(*
SPDX-FileCopyrightText: © 2026 Oleksandr Tiutyk <trofimich@gmail.com>
SPDX-License-Identifier: MIT
License: https://opensource.org/license/mit
*)

{attribute 'no_explicit_call' := 'do not call this function block directly'} 
FUNCTION_BLOCK GenericValueValidator EXTENDS Object IMPLEMENTS IGenericValueValidator
VAR
	_ClassName : STRING := __POUNAME();
	
	_TypeClass : GENERIC_TYPE_CLASS;
END_VAR

{attribute 'monitoring' := 'call'}
PROPERTY ClassName : REFERENCE TO STRING
GET
ClassName REF= _ClassName;
END_GET
END_PROPERTY

//!<param name="bInitRetains">if TRUE, the retain variables are initialized (warm start / cold start)</param>

//!<param name="bInCopyCode">if TRUE, the instance afterwards gets moved into the copy code (online change)</param>

METHOD FB_init : BOOL
VAR_INPUT
	
	bInitRetains	: BOOL;
	
	bInCopyCode	: BOOL;
	typeClass : GENERIC_TYPE_CLASS;
END_VAR
_TypeClass := typeClass;
END_METHOD

{attribute 'monitoring' := 'call'}
PROPERTY NamespaceName : REFERENCE TO STRING
GET
NamespaceName REF= CurrentNamespace.Name;
END_GET
END_PROPERTY

{attribute 'monitoring' := 'call'}
PROPERTY SelfSize : ULINT
GET
SelfSize := XSIZEOF(THIS^);
END_GET
END_PROPERTY

METHOD Validate
VAR_INPUT
	validatedObjectName : WSTRING;
END_VAR
VAR_IN_OUT CONSTANT
	valueToValidate : GENERIC_VALUE;
END_VAR
VAR
	invalidTypeException : IncompartibleGenericValueTypeException;	
END_VAR
IF valueToValidate.TypeClass <> _TypeClass THEN
	invalidTypeException.Throw(NamespaceName, ClassName, __POUNAME(), __POSITION(), validatedObjectName, valueToValidate.TypeClass, _TypeClass);
END_IF
END_METHOD

END_FUNCTION_BLOCK

(* stored: Version 1.1.0.1
   POU GenericValueValidator: Id {a6d5904d-3010-444c-98c8-80a1917cd203}, SpecialFunc None
   Property ClassName: Id {f82f2d1b-4fc3-4718-8a54-251f7a3461ed}
   Get Get: Id {f8ee5778-fbfa-4295-aae4-9ccdc19eabec}
   Method FB_init: Id {95506783-a7ce-4b15-8e1c-b1e7f4fba622}
   Property NamespaceName: Id {9a354a72-0f79-490e-939d-4595cd41c7d6}
   Get Get: Id {81f4a78c-70ec-4b46-b623-1fc67f33b3d4}
   Property SelfSize: Id {449e46a9-6074-482b-8702-4da704e912dd}
   Get Get: Id {4b470976-567f-4fd3-acda-2171efc07a0c}
   Method Validate: Id {340dfa6e-d672-4daf-b2d9-ef30de77ce10} *)
